{attribute 'linkalways'} 
{attribute 'no_explicit_call' := 'This FB is a CLASS and must be accessed using methods or properties'}
{attribute 'enable_dynamic_creation'}
FUNCTION_BLOCK _ETcVnPaddingMode EXTENDS EnumDatatypeBase
VAR
	localData : ETcVnPaddingMode;
	activeData : REFERENCE TO ETcVnPaddingMode;
	enumBaseDatatype : _DINT(localData);
END_VAR

METHOD PRIVATE AddLocalEnumeration
VAR_INPUT
	Enumeration : T_MAXSTRING;
	Value : ETcVnPaddingMode;
END_VAR
AddEnumeration(Enumeration, Value);
END_METHOD

PROPERTY PUBLIC Address : PVOID
GET
Address := ADR(activeData);
END_GET
END_PROPERTY

METHOD PUBLIC ClearReference
VAR_INPUT
END_VAR
activeData REF= localData;
SetBaseDatatypeReference();
END_METHOD

METHOD PUBLIC Clone : I_Datatype
VAR
    pClone : POINTER TO _ETcVnPaddingMode;
END_VAR
pClone := __NEW(_ETcVnPaddingMode(InitialValue := Value));
Clone := pClone^;
END_METHOD

METHOD FB_init : BOOL
VAR_INPUT
	bInitRetains : BOOL; // if TRUE, the retain variables are initialized (warm start / cold start)
	bInCopyCode : BOOL;  // if TRUE, the instance afterwards gets moved into the copy code (online change)
	InitialValue : ETcVnPaddingMode;
END_VAR
localData := InitialValue;
AddBaseDatatype(enumBaseDatatype);
ClearReference();

AddLocalEnumeration('TCVN_PM_NONE', ETcVnPaddingMode.TCVN_PM_NONE);
AddLocalEnumeration('TCVN_PM_CROP_CENTER', ETcVnPaddingMode.TCVN_PM_CROP_CENTER);
AddLocalEnumeration('TCVN_PM_LETTERBOX', ETcVnPaddingMode.TCVN_PM_LETTERBOX);
END_METHOD

PROPERTY PUBLIC Identifier : T_MAXSTRING
GET
Identifier := 'ETcVnPaddingMode';
END_GET
END_PROPERTY

METHOD IsEnumeratorValueEqual : BOOL
VAR_INPUT
	Enumerator : I_KeyValueForwardEnumerator;
END_VAR
VAR
	storedValue : ETcVnPaddingMode;
END_VAR
IF NOT Enumerator.TryGet(storedValue) THEN
	RETURN;
END_IF

IsEnumeratorValueEqual := storedValue = activeData;
END_METHOD

METHOD PUBLIC MakeReferenceTo
VAR_INPUT
	ReferenceTarget : REFERENCE TO ETcVnPaddingMode;
END_VAR
activeData REF= ReferenceTarget;
SetBaseDatatypeReference();
END_METHOD

METHOD PROTECTED SetBaseDatatypeReference
VAR_INPUT
END_VAR
enumBaseDatatype.MakeReferenceTo(activeData);
END_METHOD

PROPERTY PUBLIC Size : UDINT
GET
Size := SIZEOF(activeData);
END_GET
END_PROPERTY

METHOD TryMakeReferenceTo : BOOL
VAR_INPUT
	Target : I_Datatype;
END_VAR
VAR
	targetAsEnum : I_EnumDatatype;
	pTargetData : POINTER TO ETcVnPaddingMode;
END_VAR
IF NOT Target.TryResolveAsEnumDatatype(targetAsEnum) THEN
	RETURN;
END_IF

IF targetAsEnum.Identifier <> Identifier THEN
	RETURN;
END_IF

pTargetData := Target.Address;
activeData REF= pTargetData^;
SetBaseDatatypeReference();
TryMakeReferenceTo := TRUE;
END_METHOD

PROPERTY PUBLIC Value : ETcVnPaddingMode
GET
Value := activeData;
END_GET
SET
activeData := Value;
END_SET
END_PROPERTY

END_FUNCTION_BLOCK

(* stored: Version 1.1.0.1, ProductVersion 3.1.4024.12
   POU _ETcVnPaddingMode: Id {21ea9318-8a58-49d6-a1f3-e5760fdb1dcb}, SpecialFunc None
   Folder Constructor: Id {3564541b-070e-40f4-8ea6-c4604014473d}
   Folder Private: Id {5cd4704c-1c6e-42ec-bc88-365b64906907}
   Folder Protected: Id {a9471333-28ef-4988-8191-f9711751d7e7}
   Method AddLocalEnumeration: Id {f947a284-4f82-4357-9c92-c7f67c55e9f7}
   Property Address: Id {193a2808-d439-47e7-8a01-b35b12943323}
   Get Get: Id {e7168a7c-1971-4b2c-9738-5b735da6b4f5}
   Method ClearReference: Id {2ab4760b-c384-4ad0-a786-4f9a17e4aee0}
   Method Clone: Id {d5a82130-6115-443d-93ef-9cf9ccc93d4b}
   Method FB_init: Id {a4d24923-9389-4cff-bb1c-1d2e049e991c}
   Property Identifier: Id {f96d9860-0f07-41fd-99ac-7afb105604d1}
   Get Get: Id {41f1e3b6-6f19-4f65-a1c6-6378410829f7}
   Method IsEnumeratorValueEqual: Id {a92636eb-5451-4753-8792-91f7bc7797a7}
   Method MakeReferenceTo: Id {44f4ca8e-2a2b-4828-822a-7203eb406a20}
   Method SetBaseDatatypeReference: Id {df1155c4-9dea-4bae-9830-9208f4c613d8}
   Property Size: Id {532091b9-0c32-4ca1-8e72-755fd5d0660c}
   Get Get: Id {4e174535-8151-4787-b582-1ddf9083d69e}
   Method TryMakeReferenceTo: Id {1e61ec27-decb-4869-877e-3b8e9d691b00}
   Property Value: Id {a681233c-8bd4-4d36-9cd7-8390d339113a}
   Get Get: Id {7db50121-7eaf-4148-9f83-c135a4f09608}
   Set Set: Id {9e7c2274-c739-4168-a4c9-2978903fdb54} *)
